TYPE DUT_SERVER_SKILL_OUTPUT :
STRUCT
	///Free to use = TRUE, busy to use =FALSE
	Dummy: BOOL := TRUE;
	///Identification number of skill
	ID: UINT;
	///indentfication name of skill
	Name: STRING(80);
	///Skill activated
	Activated: BOOL;
	///Ready to do skill
	Ready: BOOL;
	///Skill in process
	Busy: BOOL;
	///Skill finish
	Done: BOOL;
	///Error in system
	Error: BOOL;
	///Range of parameters
	ParameterOutput: DUT_SERVER_PARAMETEROUTPUTARRAY;
END_STRUCT
END_TYPE

(* stored: Version 1.1.0.1, ProductVersion 3.1.0.25
   DUT DUT_SERVER_SKILL_OUTPUT: Id {239507d2-2492-4e7d-9e0a-25be0c43e887} *)
